FUNCTION_BLOCK OUT_ARRAY (* ARRAY Output to TextField *)
  (* Standard: 61499-1; Classification: GUI *)
  (* Version 0.1, 2001-05-27, JHC, Rockwell Automation, XML version with N,TYPE inputs *)
  (* Version 0.0, 1998-12-30, JHC, Rockwell Automation, Original SRC version *)
  (* Compiler header: package fb.rt.net; *)
  (* Compiler Java IBM VisualAge 3.0 *)
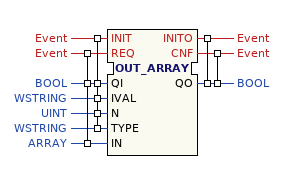
  EVENT_INPUT
    INIT WITH QI, IVAL, N, TYPE; (* Initialization *)
    REQ WITH QI, IN; (* Request *)
  END_EVENT
  EVENT_OUTPUT
    INITO WITH QO; (* Initialization Confirm *)
    CNF WITH QO; (* Service Confirmation *)
  END_EVENT
  VAR_INPUT
    QI : BOOL; (* Input event qualifier *)
    IVAL : WSTRING; (* Initial contents *)
    N : UINT; (* Number of array elements *)
    TYPE : WSTRING; (* Array element type *)
    IN : ARRAY; (* Output value *)
  END_VAR
  VAR_OUTPUT
    QO : BOOL; (* Output event qualifier *)
  END_VAR
END_FUNCTION_BLOCK
